{attribute 'hide_all_locals'}
FUNCTION_BLOCK AxesReset IMPLEMENTS ITask
VAR_INPUT
END_VAR
VAR_OUTPUT
END_VAR
VAR
	resetMover : Tc2_MC2.MC_Reset;
	_axis : REFERENCE TO Tc2_MC2.AXIS_REF;
	_ResetMover : BOOL;
	state : INT;
	_busy : BOOL;
	_error : BOOL;
	_done : BOOL;
END_VAR

CASE State OF
	0:
		IF _ResetMover THEN
			_done := FALSE;
			_error := FALSE;
			_busy := TRUE;
			resetMover.Execute := TRUE;
			IF resetMover.Busy THEN
				State := 10;
				_ResetMover := FALSE;
			END_IF
		END_IF
	
	10:
		IF NOT resetMover.Busy THEN
			IF resetMover.Done THEN
				_done := TRUE;
			ELSIF resetMover.Error THEN
				_error := TRUE;
			END_IF
			_busy := FALSE;
			resetMover.Execute := FALSE;
			State := 0;
		END_IF
END_CASE

resetMover(Axis := _axis);

{warning 'add method implementation '}
METHOD Abort : BOOL
resetMover.Execute := FALSE;
_busy := FALSE;
_ResetMover := FALSE;
Abort := TRUE;
State := 0;
END_METHOD

{warning 'add property implementation'}
PROPERTY Busy : BOOL
GET
Busy := _busy;
END_GET
END_PROPERTY

{warning 'add property implementation'}
PROPERTY Done : BOOL
GET
Done := _done;
END_GET
END_PROPERTY

{warning 'add property implementation'}
PROPERTY Error : BOOL
GET
Error := _error;
END_GET
END_PROPERTY

METHOD Execute : BOOL
VAR_INPUT
END_VAR
Execute := _ResetMover := true;
END_METHOD

METHOD FB_init : BOOL
VAR_INPUT
	bInitRetains : BOOL; // if TRUE, the retain variables are initialized (warm start / cold start)
	bInCopyCode : BOOL;  // if TRUE, the instance afterwards gets moved into the copy code (online change)
	axis : reference TO AXIS_REF;
END_VAR
_axis REF= axis;
END_METHOD

END_FUNCTION_BLOCK

(* stored: Version 1.1.0.1, ProductVersion 3.1.4024.6
   POU AxesReset: Id {19c7231b-8311-413c-9d34-e6adc74e815f}, SpecialFunc None
   Method Abort: Id {9e36c0f1-29b1-495e-81a0-1b56d8641dad}
   Property Busy: Id {4bd0c1bc-04e3-4035-be20-37a4a7951312}
   Get Get: Id {10088129-c3bc-45c5-a92a-560ec05cd1e0}
   Property Done: Id {69a4036c-fbd6-447e-9a81-2a36e44fa345}
   Get Get: Id {de08bd98-cb25-4cfe-9549-e45117710413}
   Property Error: Id {eb85cd05-7c9e-445c-a5b5-cee06b091b11}
   Get Get: Id {5d4ec38d-ee89-4e4f-952f-381714593cd5}
   Method Execute: Id {970be4f7-baea-484f-958b-1c0a16dff6a0}
   Method FB_init: Id {6e3c62b3-f95b-43c4-9b6d-e9f710b1d755} *)
